// TIA Portal V19 export
TYPE "typePressureGuageRs485ControlNodeMonitoring"
TITLE = LBC_typeAnalogOutputControlNodeMonitoring
// Control Node Wapper monitoring values
// stored: Access Published
   STRUCT
      valid { ExternalAccessible := 'False'; ExternalVisible := 'False'; ExternalWritable := 'False'} : Bool;   // Valid set of output values available at the FB
      busy { ExternalAccessible := 'False'; ExternalVisible := 'False'; ExternalWritable := 'False'} : Bool;   // Working and new output values can be expected
      error { ExternalAccessible := 'False'; ExternalVisible := 'False'; ExternalWritable := 'False'} : Bool;   // An error occurred during the execution of the FB
      status { ExternalAccessible := 'False'; ExternalVisible := 'False'; ExternalWritable := 'False'} : Word;   // 16#0000-16#7FFF: Status of the FB 16#8000-16#FFFF: Error identification (see following Table)
      limitHigh2 { ExternalAccessible := 'False'; ExternalVisible := 'False'; ExternalWritable := 'False'} : Bool;   // Limit high 2 exceeded (Lim 2 > Lim1, resets Lim 1)
      limitHigh1 { ExternalAccessible := 'False'; ExternalVisible := 'False'; ExternalWritable := 'False'} : Bool;   // Limit high 1 exceeded
      limitLow1 { ExternalAccessible := 'False'; ExternalVisible := 'False'; ExternalWritable := 'False'} : Bool;   // Limit low 1 exceeded
      limitLow2 { ExternalAccessible := 'False'; ExternalVisible := 'False'; ExternalWritable := 'False'} : Bool;   // Limit low 2 exceeded (Lim 2 < Lim1, resets Lim 1)
      maxValueReached { ExternalAccessible := 'False'; ExternalVisible := 'False'; ExternalWritable := 'False'} : Bool;   // Maximum configured process value reached. Value is limited to the maximum configured value.
      minValueReached { ExternalAccessible := 'False'; ExternalVisible := 'False'; ExternalWritable := 'False'} : Bool;   // Minimum configured process value reached. Value is limited to the minimum configured value.
   END_STRUCT;
END_TYPE
